FUNCTION_BLOCK TcoToggleTaskTests EXTENDS TcoCore.TcoToggleTask
VAR
    _isOn : BOOL;
    _isOff : BOOL;
    _isEnabled : BOOL;
    _isToggleRequestTrue : BOOL;
    _counterValue : ULINT;
    _counterValuePV : ULINT;
    _toggleCounter : ULINT;
    _runCounter : ULINT;
    _onFtrigCounter : ULINT;
    _onRtrigCounter : ULINT;
    _onCounter : ULINT;
    _offCounter : ULINT;
    _onStateChangeCounter : ULINT;
    _taskOnCounter : ULINT;
    _taskOffCounter : ULINT;
    _stateChangedCounter : ULINT;
    _previousState : BOOL;
    _myIdentity : ULINT;
    _myContextIdentity : ULINT;
    _myContextStartCount : ULINT;
    _myContextEndCount : ULINT;
    _myParentIdentity : ULINT;
END_VAR

ExecutionBody();

METHOD INTERNAL Disable
THIS^.Enabled := FALSE;
END_METHOD

METHOD INTERNAL Enable
THIS^.Enabled := TRUE;
END_METHOD

{attribute 'TcRpcEnable'}
METHOD INTERNAL ExecutionBody
Run();
_runCounter := _runCounter + 1;

IF _previousState <> THIS^.State THEN
    _stateChangedCounter := _stateChangedCounter + 1;
END_IF;

_previousState := THIS^.State;
END_METHOD

{attribute 'TcRpcEnable'}
METHOD INTERNAL GetMessage : STRING
GetMessage := SUPER^._messenger._mime.Text;
END_METHOD

METHOD PROTECTED Main
VAR
END_VAR
END_METHOD

(*~
    <docu>
        <summary>
            Executes when toggle task changes its state from '''TRUE''' to '''FALSE'''.
        </summary>
    </docu>
~*)
METHOD PROTECTED OnFtrig
_onFtrigCounter := _onFtrigCounter + 1;
END_METHOD

(*~
    <docu>
        <summary>
            Executes when toggle task changes its state from '''FALSE''' to '''TRUE'''.
        </summary>
    </docu>
~*)
METHOD PROTECTED OnRtrig
_onRtrigCounter := _onRtrigCounter + 1;
END_METHOD

(*~
    <docu>
        <summary>
            Executes when toggle task changes its state .
        </summary>
    </docu>
~*)
METHOD PROTECTED OnStateChange
_onStateChangeCounter := _onStateChangeCounter + 1;
END_METHOD

{attribute 'TcRpcEnable'}
METHOD INTERNAL PostMessage
VAR_INPUT
    Message : STRING;
END_VAR
THIS^.Messenger.Post(Message, eMessageCategory.Error);
END_METHOD

{attribute 'TcRpcEnable'}
METHOD INTERNAL ReadOutIdentities
_myIdentity := THIS^.Identity;
_myContextIdentity := THIS^.Context.Identity;
_myContextStartCount := THIS^.Context.StartCycleCount;
_myContextEndCount := THIS^.Context.EndCycleCount;
_myParentIdentity := THIS^.Parent.Identity;
END_METHOD

{attribute 'TcRpcEnable'}
METHOD INTERNAL ReadOutState
_isOn := THIS^.IsOn;
_isOff := THIS^.IsOff;
_isEnabled := THIS^.Enabled;
_isToggleRequestTrue := THIS^._toggleRequest;
END_METHOD

{attribute 'TcRpcEnable'}
METHOD INTERNAL SetPreviousState
VAR_INPUT
    inValue : BOOL;
END_VAR
THIS^._previousState := inValue;
END_METHOD

{attribute 'TcRpcEnable'}
METHOD INTERNAL SetState
VAR_INPUT
    inState : BOOL;
END_VAR
THIS^._state := inState;
END_METHOD

{attribute 'TcRpcEnable'}
METHOD INTERNAL SetToggleRequest
THIS^._toggleRequest := TRUE;
END_METHOD

(*~
    <docu>
        <summary>
            Executes when toggle task is in ```Off``` state .
        </summary>
    </docu>
~*)
METHOD PROTECTED TaskOff
_taskOffCounter := _taskOffCounter + 1;
_counterValue := _counterValue - 1;
_CounterValuePV := _counterValue;
END_METHOD

(*~
    <docu>
        <summary>
            Executes when toggle task is in  ```On``` state .
        </summary>
    </docu>
~*)
METHOD PROTECTED TaskOn
_taskOnCounter := _taskOnCounter + 1;
_counterValue := _counterValue + 1;
_CounterValuePV := _counterValue;
END_METHOD

{attribute 'TcRpcEnable'}
METHOD INTERNAL TriggerOff
THIS^.Off();
_offCounter := _offCounter + 1;
END_METHOD

{attribute 'TcRpcEnable'}
METHOD INTERNAL TriggerOn
THIS^.On();
_onCounter := _onCounter + 1;
END_METHOD

{attribute 'TcRpcEnable'}
METHOD INTERNAL TriggerToggle
THIS^.Toggle();
_toggleCounter := _toggleCounter + 1;
END_METHOD

END_FUNCTION_BLOCK

(* stored: Version 1.1.0.1
   POU TcoToggleTaskTests: Id {772d1beb-fd7c-03c3-2489-a6c5d7a9708c}, SpecialFunc None
   Method Disable: Id {268f2058-6aa2-0bc9-3e41-8eb17a9ec731}
   Method Enable: Id {0f5509ed-673e-05be-0f08-2878d85be3da}
   Method ExecutionBody: Id {d2c08234-959e-00a3-2cf0-7764ba6fd8e2}
   Method GetMessage: Id {e7526a03-c3c0-0e86-2c05-862603a5c6c5}
   Method Main: Id {244a78f8-0b46-0493-2393-a6c8a05c4da0}
   Method OnFtrig: Id {81f92352-91b8-0d38-1074-6f2338d59118}
   Method OnRtrig: Id {75c359b2-0c9e-0c8b-05e1-282cf5bcb466}
   Method OnStateChange: Id {7374d645-e61b-0291-1c70-20fd2c77b62a}
   Method PostMessage: Id {c90282f7-bce9-0465-20e7-e8f7de390f10}
   Method ReadOutIdentities: Id {d29521d2-6f84-0538-2f15-11e2cb62edda}
   Method ReadOutState: Id {08e54675-4b27-0c1a-21b6-6bada9936a11}
   Method SetPreviousState: Id {dd0bedf4-4080-099f-0411-61a004a324a0}
   Method SetState: Id {c4f8f908-a29e-078f-3f47-8e3dc55c1fdd}
   Method SetToggleRequest: Id {2f9e9a28-57e0-0be8-369d-ae13d5145ac8}
   Method TaskOff: Id {7c9900ff-df50-0145-2e9c-02b73c53bfbb}
   Method TaskOn: Id {7b97312c-442f-0516-281c-cfac93831dd7}
   Method TriggerOff: Id {c9e02822-ae4f-075b-0744-a39394f45bb6}
   Method TriggerOn: Id {3d75fcb9-2c68-0f2b-0937-2bb7dee18863}
   Method TriggerToggle: Id {4226c295-2f1b-0597-1199-477276f01c63} *)
